(*

.. <legal notes>

legal notes
=================
| SPDX-FileCopyrightText: © 2026 Oleksandr Tiutyk <trofimich@gmail.com>
| SPDX-License-Identifier: LGPL-3.0-only
| For details check: LGPL-3.0-only_

.. _LGPL-3.0-only: https://www.gnu.org/licenses/lgpl-3.0.en.html

.. </legal notes>

*)

{attribute 'no_explicit_call' := 'Direct call is not allowed'} 
PROGRAM Memory
VAR
	_ClassName : STRING := __POUNAME();
END_VAR

{attribute 'monitoring' := 'call'}
PROPERTY ClassName : STRING
GET
ClassName := _ClassName;
END_GET
END_PROPERTY

METHOD GetAddressFromInterface : PVOID
VAR_INPUT
	interfaceInstance : __SYSTEM.IQueryInterface; 
END_VAR
VAR
	interfacePointer : POINTER TO PVOID;
END_VAR
IF interfaceInstance <> 0 THEN
	interfacePointer := ADR(interfaceInstance);
	
	GetAddressFromInterface := interfacePointer^ - XSIZEOF(interfaceInstance);	
END_IF
END_METHOD

METHOD IsDynamicData : BOOL
VAR_INPUT
	dataAddress : PVOID;
	dataSize : UDINT := 1;
END_VAR
IsDynamicData := Tc2_System.F_CheckMemoryArea(dataAddress, dataSize) = E_TcMemoryArea.Dynamic;
END_METHOD

{attribute 'monitoring' := 'call'}
PROPERTY NamespaceName : STRING
GET
NamespaceName := CurrentNamespace.Name;
END_GET
END_PROPERTY

METHOD TryReleaseDynamicMemory : BOOL
VAR_IN_OUT
	address : POINTER TO BYTE;	
END_VAR
VAR_INPUT
	isObject : BOOL;
END_VAR
VAR
	objectPointer : POINTER TO Object;
	objectClassName : STRING;
END_VAR
IF address = 0 OR_ELSE NOT Memory.IsDynamicData(address, 1) THEN
	RETURN;
END_IF

IF isObject THEN
	objectPointer := address;
	objectClassName := objectPointer^.ClassName;
	
	__DELETE(objectPointer);
	address := 0;
	
	LogManager.TryLogMessage(WideStrings.Concat255("Object of class '", TO_WSTRING(objectClassName), "' disposed at ", TO_WSTRING(SystemDateTimeManager.SystemLocalDateTime)), LOG_CATEGORY.INFORMATION, TO_WSTRING(ClassName), "ReleaseDynamicMemory", "ObjectDispose");
ELSE
	__DELETE(address);
END_IF

TryReleaseDynamicMemory := TRUE;
END_METHOD

METHOD TryReleaseDynamicObject : BOOL
VAR_IN_OUT
	instance : IObject;	
END_VAR
VAR
	objectPointer : POINTER TO Object;
END_VAR
IF instance = 0 THEN
	RETURN;
END_IF
	
objectPointer := instance.SelfAddress;

TryReleaseDynamicObject := TryReleaseDynamicMemory(objectPointer, TRUE);

IF TryReleaseDynamicObject THEN
	instance := 0;
END_IF
END_METHOD

END_PROGRAM

(* stored: Version 1.1.0.1
   POU Memory: Id {cb04704d-a05c-4735-b40b-67a92f3f86d5}, SpecialFunc None
   Property ClassName: Id {f0cb7e04-3fa7-438c-9fb8-38f358e717d9}
   Get Get: Id {9465e911-db84-4abe-a766-2f2cfe6e21d4}
   Method GetAddressFromInterface: Id {6158ab88-0c76-435a-bca8-37fff74aaa20}
   Method IsDynamicData: Id {4c5114c7-cc73-448a-9f8f-fa67bfde37e3}
   Property NamespaceName: Id {5aeb5d90-3cbf-4d4b-8537-6b3b6ccb7bea}
   Get Get: Id {464e75ad-f0ba-4929-8b1e-1713c91d4754}
   Method TryReleaseDynamicMemory: Id {5fe5bc2a-b608-418e-9ff0-e9c1a91c92f5}
   Method TryReleaseDynamicObject: Id {1a29f8e6-f929-40c9-bee2-ed6219c50a45} *)
